{attribute 'qualified_only'}
VAR_GLOBAL
	distanceToMirror : REAL;    // Distance between user and mirror in meters
    lightStatus : BOOL := FALSE;   // Light status (ON/OFF)
    timerActive : BOOL := FALSE;   // Timer active status
    timerElapsed : BOOL := FALSE;  // Timer finished status
END_VAR

(* stored: Version 1.1.0.1, ProductVersion 3.1.4024.12
   GVL GVL: Id {ef4b1691-91bd-4796-b076-91122cad1d34} *)
